// TIA Portal V19 export
DATA_BLOCK "DB_Temporaer"   // DB999
{ S7_Optimized_Access := 'TRUE' }
// stored: AutoNumber false, MemoryReserve 100
   VAR RETAIN
      Drucksensoren_deaktiviert : Bool;   // 20.01.22
   END_VAR
BEGIN
END_DATA_BLOCK
